//{attribute 'qualified_only'}
{attribute 'strict'}
TYPE eDeffuzyMethod :
(
	Centroid
);
END_TYPE

(* stored: Version 1.1.0.1, ProductVersion 3.1.4024.6
   DUT eDeffuzyMethod: Id {8d399c7b-8798-4530-9587-52750ef778d9} *)
